FUNCTION_BLOCK FINAL FB_SystemEvent EXTENDS FB_EventLogger
VAR_INPUT
	Raise					: BOOL;	     				//Event Raiser
	EventType				: E_EventType;				//Event Type Enum 
	EventEntry				: TcEventEntry;				//Event Entry 
	Arg0					: STRING := '';				//Event Argument {0}
	Arg1					: STRING := '';				//Event Argument {1}
	Arg2					: STRING := '';				//Event Argument {2}
END_VAR
VAR_IN_OUT
	Control					: ST_System;				//Machine Control Instance
END_VAR
VAR           
	_EventTimer_ET			: REAL;						//Event timer elapsed
	_Alarm					: BOOL;						//Device Alarm
	_Warning				: BOOL;						//Device Warning
END_VAR
VAR PERSISTENT
	_AlarmMute				: BOOL;						//Event Mute
	_EventTimer_PT			: REAL;						//Event timer preset time
END_VAR

IF NOT _AlarmMute AND NOT Control.Inputs.AlarmAck.Enabled THEN
	IF Raise THEN
		_EventTimer_ET :=  _EventTimer_ET + Control.SystemTime.ScanTime;
	END_IF
END_IF

CASE EventType OF
	E_EventType.eAlarm:
		M_LogAlarm(Execute:= _EventTimer_ET > _EventTimer_PT , Arg0:= Arg0, Arg1:= Arg1, Arg2:= Arg2, EventEntry:= EventEntry,Clear:= NOT _Alarm, Message:= Control.Outputs.AlarmMessage);
		IF _EventTimer_ET > _EventTimer_PT THEN
			IF NOT Control.Outputs.Alarm THEN 
				Control.Outputs.Alarm := TRUE;
			END_IF		
			_Alarm := TRUE;
		END_IF
	E_EventType.eWarning:
		M_LogWarning(Execute:= _EventTimer_ET > _EventTimer_PT , Arg0:= Arg0, Arg1:= Arg1, Arg2:= Arg2, EventEntry:= EventEntry,Clear := NOT _Warning,Message:= Control.Outputs.WarningMessage);
		IF _EventTimer_ET > _EventTimer_PT THEN
			IF NOT Control.Outputs.Warning THEN 
				Control.Outputs.Warning := TRUE;
			END_IF		
			_Warning := TRUE;
		END_IF
	E_EventType.eAlert:
		M_LogAlert(Execute:= Raise, Arg0:= Arg0, Arg1:= Arg1, Arg2:= Arg2, EventEntry:= EventEntry, Message:= Control.Outputs.AlertMessage);
		IF NOT Control.Outputs.Alert AND Raise THEN
			Control.Outputs.Alert := TRUE;
		END_IF
	E_EventType.eMessage:
		M_LogMessage(Execute:= Raise, Arg0:= Arg0, Arg1:= Arg1, Arg2:= Arg2, EventEntry:= EventEntry);
	ELSE
		RETURN;

END_CASE

IF NOT Raise  OR _AlarmMute OR Control.Inputs.AlarmAck.Enabled THEN
	 _EventTimer_ET := 0;_Alarm := FALSE;_Warning := FALSE;
END_IF

{attribute 'monitoring' := 'variable'}
PROPERTY PUBLIC Alarm : Bool
GET
Alarm := _Alarm;
END_GET
END_PROPERTY

{attribute 'monitoring' := 'variable'}
PROPERTY PUBLIC AlarmMute : BOOL
SET
AlarmMute := _AlarmMute;
END_SET
END_PROPERTY

{attribute 'monitoring' := 'variable'}
PROPERTY PUBLIC EventTimer_ET : real
GET
EventTimer_ET := _EventTimer_ET;
END_GET
END_PROPERTY

{attribute 'monitoring' := 'variable'}
PROPERTY PUBLIC EventTimer_PT : real
GET
EventTimer_PT := _EventTimer_PT;
END_GET
SET
_EventTimer_PT := EventTimer_PT;
END_SET
END_PROPERTY

{attribute 'monitoring' := 'variable'}
PROPERTY PUBLIC Warning : Bool
GET
Warning := _Warning;
END_GET
END_PROPERTY

END_FUNCTION_BLOCK

(* stored: Version 1.1.0.1, ProductVersion 3.1.4024.3
   POU FB_SystemEvent: Id {c145d96a-3e91-45f3-a18f-80f040a4f6f7}, SpecialFunc None
   Property Alarm: Id {7708bd8f-23bd-4e4e-b0c3-dff049aa72f9}
   Get Get: Id {f942402f-f875-4ab3-8029-85c3a58b4a8c}
   Property AlarmMute: Id {e633d145-59f8-44ee-8097-452d3869313d}
   Set Set: Id {f0f3aa87-bffc-4a45-b2ad-7af035050a29}
   Property EventTimer_ET: Id {ba85efe3-bf77-4ce9-b51c-faf44194650f}
   Get Get: Id {65018f71-d8a2-454d-896e-4f4d948fa3f5}
   Property EventTimer_PT: Id {d78a4612-36c8-4fd4-b744-c20aca951619}
   Get Get: Id {ff604f1e-1b15-47d5-a466-7fb31c99ff91}
   Set Set: Id {e95157f9-6d51-45ab-b59a-9da1695f28c0}
   Property Warning: Id {4525ad36-95fa-4e77-9aad-f6596211ab76}
   Get Get: Id {88ac7baa-81b9-4ee6-b0c9-3b978aa092c3} *)
